// Mitsubishi GX Works2 project: PLC 특수기능 (Line Pulse)   PLC: Q03UDV

PROGRAM MAIN
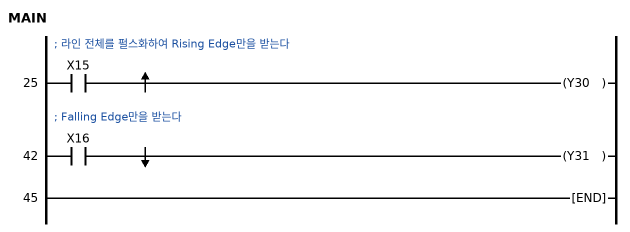
; 라인 전체를 펄스화하여 Rising Edge만을 받는다
25    LD      X15
      MEP
      OUT     Y30
; Falling Edge만을 받는다
42    LD      X16
      MEF
      OUT     Y31
45    END
END_PROGRAM
